// SIMATIC S7-200 project (STEP 7-Micro/WIN), CPU 224XP CN REL 02.01

SYMBOL_TABLE USER1
M_Main_Green     M0.0
M_Main_Yellow    M0.1
M_Main_Red       M0.2
M_Sp_Green       M0.3
M_Sp_Yellow      M0.4
M_Sp_Red         M0.5
O_Main_Green     Q0.0
O_Main_Yellow    Q0.1
O_Main_Red       Q0.2
O_Sp_Green       Q0.3
O_Sp_Yellow      Q0.4
O_Sp_Red         Q0.5
Start_Pause      I0.0
Reset            I0.1
Counter          VW0
MODDONE          M1.0
MODERR           MB2
MODSDONE         M1.1
MODSERR          MB4
Q_Start_Pause    Q0.6
END_SYMBOL_TABLE

SYMBOL_TABLE S7-200 符号
Always_On        SM0.0    // 始终接通为 ON
First_Scan_On    SM0.1    // 仅第一个扫描周期中接通为 ON
Clock_1s         SM0.5    // 在 1 秒钟的循环周期内，接通为 ON 0.5 秒，关断为 OFF 0.5  秒
END_SYMBOL_TABLE

ORGANIZATION_BLOCK MAIN:OB1
TITLE=PROGRAM COMMENTS
BEGIN
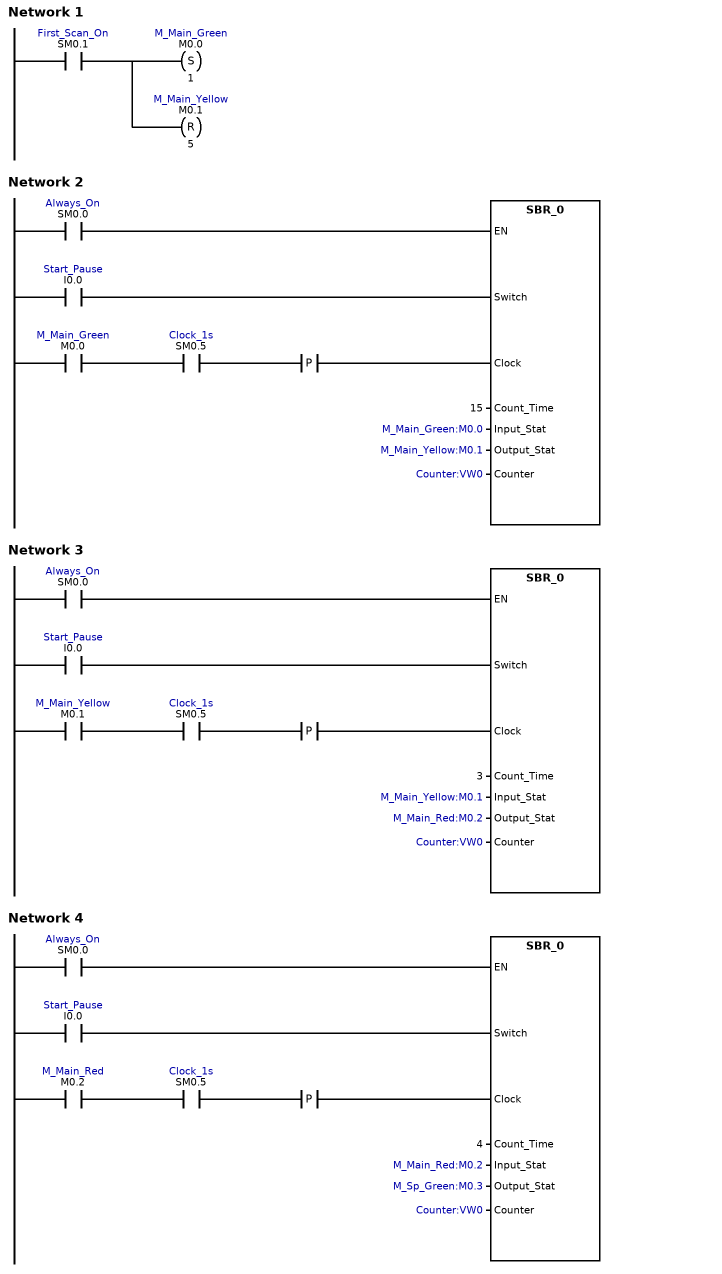
Network 1
LD     First_Scan_On:SM0.1
S      M_Main_Green:M0.0, 1
R      M_Main_Yellow:M0.1, 5
Network 2
LD     Always_On:SM0.0
=      L60.0
LD     Start_Pause:I0.0
=      L63.7
LD     M_Main_Green:M0.0
A      Clock_1s:SM0.5
EU
=      L63.6
LD     L60.0
CALL   SBR_0:SBR0, L63.7, L63.6, 15, M_Main_Green:M0.0, M_Main_Yellow:M0.1, Counter:VW0
Network 3
LD     Always_On:SM0.0
=      L60.0
LD     Start_Pause:I0.0
=      L63.7
LD     M_Main_Yellow:M0.1
A      Clock_1s:SM0.5
EU
=      L63.6
LD     L60.0
CALL   SBR_0:SBR0, L63.7, L63.6, 3, M_Main_Yellow:M0.1, M_Main_Red:M0.2, Counter:VW0
Network 4
LD     Always_On:SM0.0
=      L60.0
LD     Start_Pause:I0.0
=      L63.7
LD     M_Main_Red:M0.2
A      Clock_1s:SM0.5
EU
=      L63.6
LD     L60.0
CALL   SBR_0:SBR0, L63.7, L63.6, 4, M_Main_Red:M0.2, M_Sp_Green:M0.3, Counter:VW0
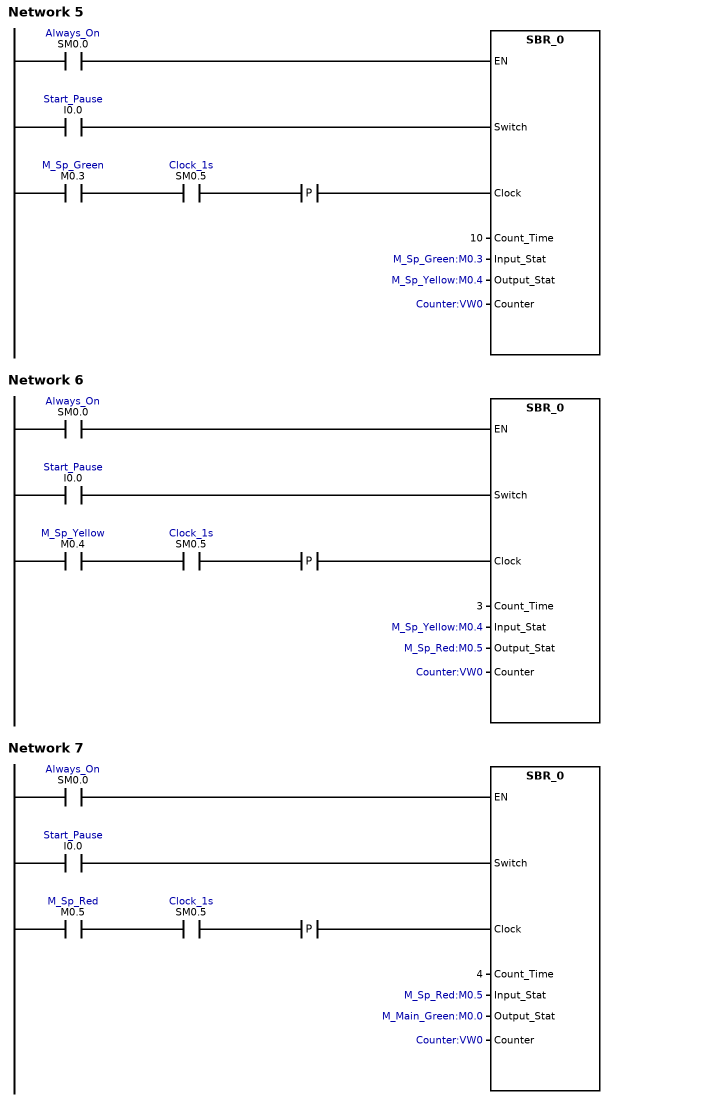
Network 5
LD     Always_On:SM0.0
=      L60.0
LD     Start_Pause:I0.0
=      L63.7
LD     M_Sp_Green:M0.3
A      Clock_1s:SM0.5
EU
=      L63.6
LD     L60.0
CALL   SBR_0:SBR0, L63.7, L63.6, 10, M_Sp_Green:M0.3, M_Sp_Yellow:M0.4, Counter:VW0
Network 6
LD     Always_On:SM0.0
=      L60.0
LD     Start_Pause:I0.0
=      L63.7
LD     M_Sp_Yellow:M0.4
A      Clock_1s:SM0.5
EU
=      L63.6
LD     L60.0
CALL   SBR_0:SBR0, L63.7, L63.6, 3, M_Sp_Yellow:M0.4, M_Sp_Red:M0.5, Counter:VW0
Network 7
LD     Always_On:SM0.0
=      L60.0
LD     Start_Pause:I0.0
=      L63.7
LD     M_Sp_Red:M0.5
A      Clock_1s:SM0.5
EU
=      L63.6
LD     L60.0
CALL   SBR_0:SBR0, L63.7, L63.6, 4, M_Sp_Red:M0.5, M_Main_Green:M0.0, Counter:VW0
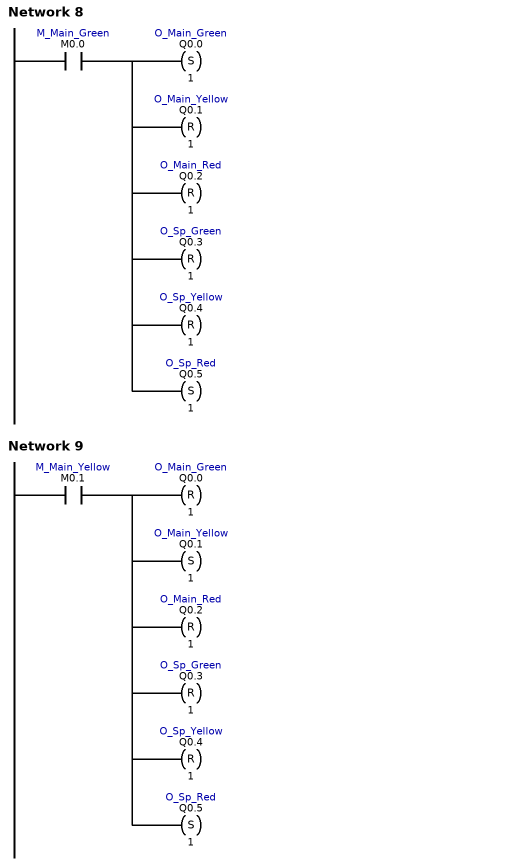
Network 8
LD     M_Main_Green:M0.0
S      O_Main_Green:Q0.0, 1
R      O_Main_Yellow:Q0.1, 1
R      O_Main_Red:Q0.2, 1
R      O_Sp_Green:Q0.3, 1
R      O_Sp_Yellow:Q0.4, 1
S      O_Sp_Red:Q0.5, 1
Network 9
LD     M_Main_Yellow:M0.1
R      O_Main_Green:Q0.0, 1
S      O_Main_Yellow:Q0.1, 1
R      O_Main_Red:Q0.2, 1
R      O_Sp_Green:Q0.3, 1
R      O_Sp_Yellow:Q0.4, 1
S      O_Sp_Red:Q0.5, 1
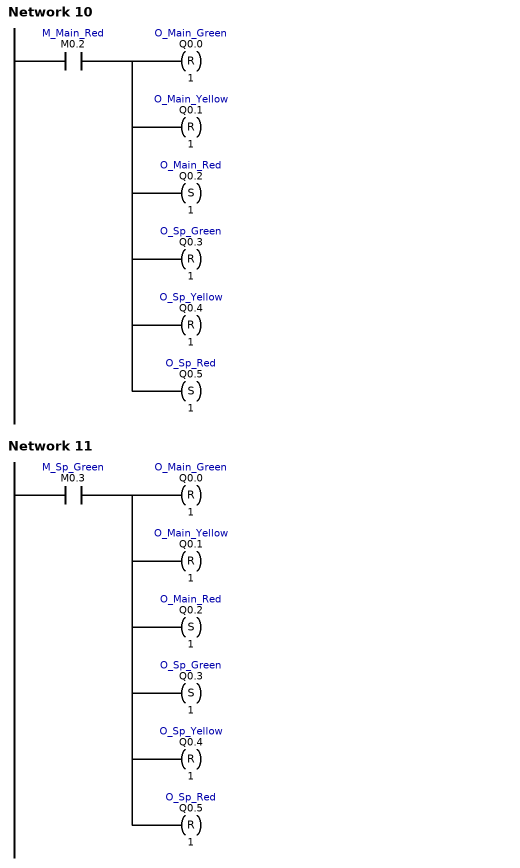
Network 10
LD     M_Main_Red:M0.2
R      O_Main_Green:Q0.0, 1
R      O_Main_Yellow:Q0.1, 1
S      O_Main_Red:Q0.2, 1
R      O_Sp_Green:Q0.3, 1
R      O_Sp_Yellow:Q0.4, 1
S      O_Sp_Red:Q0.5, 1
Network 11
LD     M_Sp_Green:M0.3
R      O_Main_Green:Q0.0, 1
R      O_Main_Yellow:Q0.1, 1
S      O_Main_Red:Q0.2, 1
S      O_Sp_Green:Q0.3, 1
R      O_Sp_Yellow:Q0.4, 1
R      O_Sp_Red:Q0.5, 1
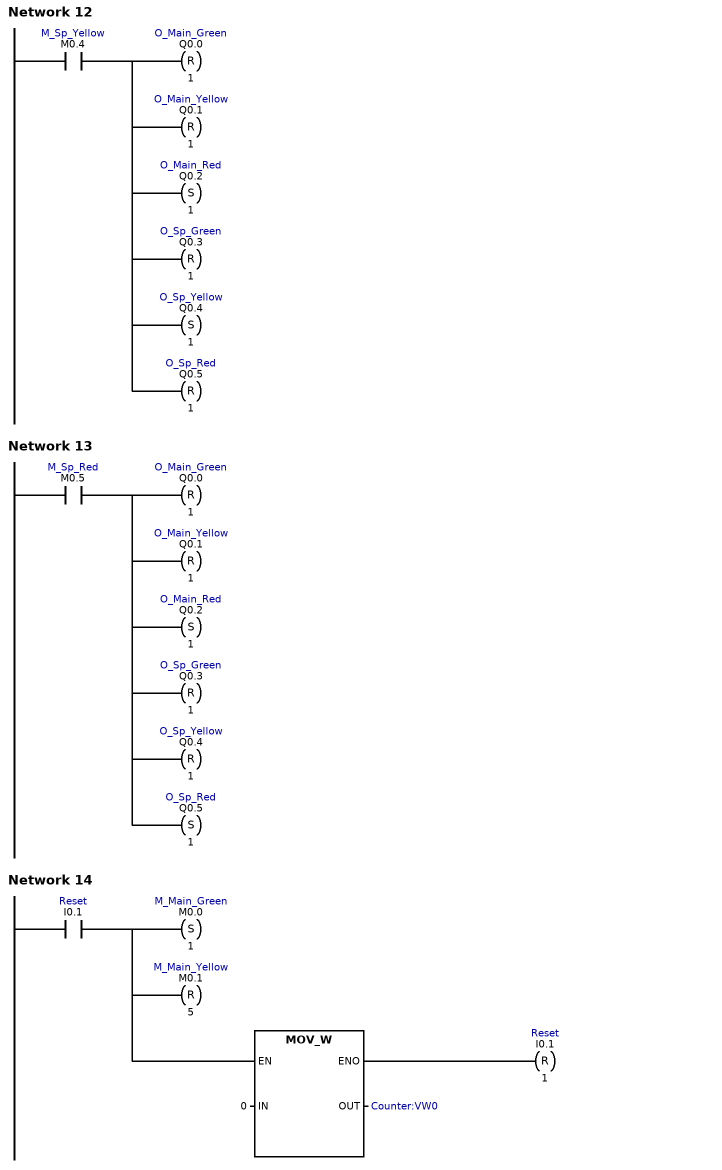
Network 12
LD     M_Sp_Yellow:M0.4
R      O_Main_Green:Q0.0, 1
R      O_Main_Yellow:Q0.1, 1
S      O_Main_Red:Q0.2, 1
R      O_Sp_Green:Q0.3, 1
S      O_Sp_Yellow:Q0.4, 1
R      O_Sp_Red:Q0.5, 1
Network 13
LD     M_Sp_Red:M0.5
R      O_Main_Green:Q0.0, 1
R      O_Main_Yellow:Q0.1, 1
S      O_Main_Red:Q0.2, 1
R      O_Sp_Green:Q0.3, 1
R      O_Sp_Yellow:Q0.4, 1
S      O_Sp_Red:Q0.5, 1
Network 14
LD     Reset:I0.1
S      M_Main_Green:M0.0, 1
R      M_Main_Yellow:M0.1, 5
MOVW   0, Counter:VW0
AENO
R      Reset:I0.1, 1
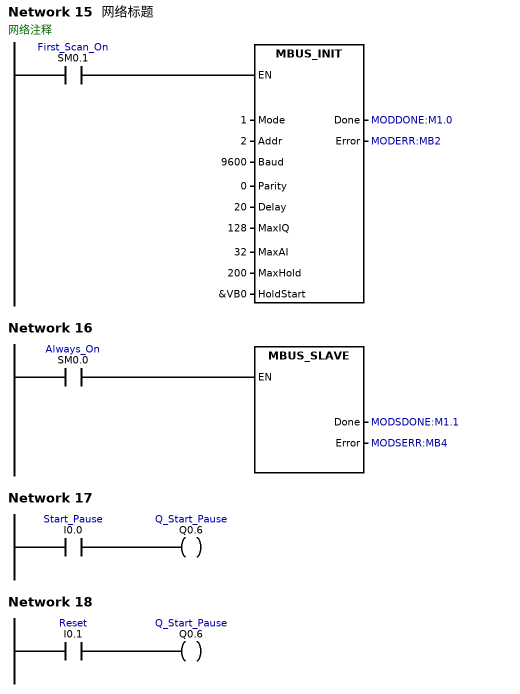
Network 15 // 网络标题
// 网络注释
LD     First_Scan_On:SM0.1
CALL   MBUS_INIT:SBR1, 1, 2, 9600, 0, 20, 128, 32, 200, &VB0, MODDONE:M1.0, MODERR:MB2
Network 16
LD     Always_On:SM0.0
CALL   MBUS_SLAVE:SBR2, MODSDONE:M1.1, MODSERR:MB4
Network 17
LD     Start_Pause:I0.0
=      Q_Start_Pause:Q0.6
Network 18
LD     Reset:I0.1
=      Q_Start_Pause:Q0.6
END_ORGANIZATION_BLOCK

SUBROUTINE_BLOCK SBR_0:SBR0
TITLE=SUBROUTINE COMMENTS
VAR_INPUT
Switch:BOOL;	// L0.0 
Clock:BOOL;	// L0.1 
Count_Time:INT;	// LW1 
END_VAR
VAR_IN_OUT
Input_Stat:BOOL;	// L3.0 
Output_Stat:BOOL;	// L3.1 
Counter:INT;	// LW4 
END_VAR
BEGIN
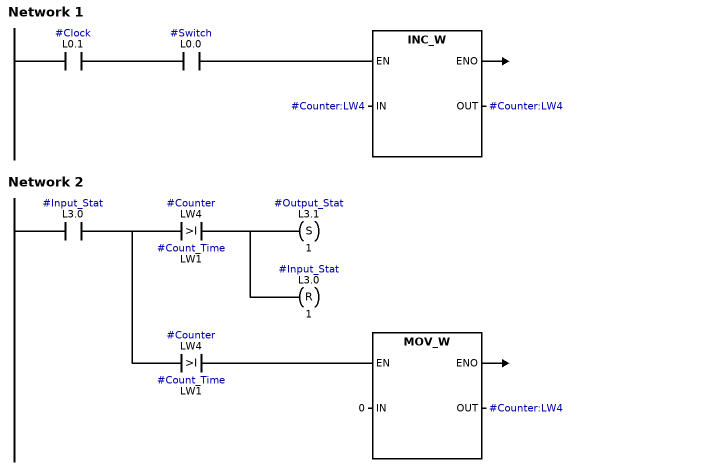
Network 1
LD     #Clock:L0.1
A      #Switch:L0.0
INCW   #Counter:LW4
Network 2
LD     #Input_Stat:L3.0
LPS
AW>    #Counter:LW4, #Count_Time:LW1
S      #Output_Stat:L3.1, 1
R      #Input_Stat:L3.0, 1
LPP
AW>    #Counter:LW4, #Count_Time:LW1
MOVW   0, #Counter:LW4
END_SUBROUTINE_BLOCK

// SBR1: protected block, not included

// SBR2: protected block, not included

// SBR3: protected block, not included
